PROGRAM PRG_SysPulses
VAR 
// 50% Duty Cycle
	fbXO_250Hz    		:FB_Pulse;	//Correct at 2ms tick
	fbXO_50Hz     		:FB_Pulse;	//Correct at 2ms tick
	fbXO_10Hz			:FB_Pulse;	//Correct at 2ms tick
	fbXO_5Hz			:FB_Pulse;	//Correct at 2ms tick
	fbXO_2Hz			:FB_Pulse;	//Correct at 2ms tick	
	fbXO_1Hz			:FB_Pulse;	//Correct at 2ms tick
	fbXO_05Hz			:FB_Pulse;	//Correct at 2ms tick
	// Frictions
	fbXO_1p85Hz			:FB_Pulse;	//Correct at 2ms tick
	fbXO_1p52Hz			:FB_Pulse;	//Correct at 2ms tick
	fbXO_1p33Hz			:FB_Pulse;	//Correct at 2ms tick
	fbXO_1p19Hz			:FB_Pulse;	//Correct at 2ms tick	
	
// 70/30 Duty Cycle
	fbXO_1Hz_7030		:FB_Pulse;	//Correct at 2ms tick
	
// 80/20 Duty Cycle
	fbXO_1Hz_8020		:FB_Pulse;	//Correct at 2ms tick
//-----------------------------------------------oldschoo1		
END_VAR

(*** Oscilator Pulse Generators at 2ms tick ***)

// 50% Duty Cycle
	fbXO_250Hz(
		bEnable				:=	TRUE,
		tPulseOn			:=	T#2MS,
		tPulseOff			:=	T#2MS,
		bFlash				=>	bFlash250Hz);
	fbXO_50Hz( 
		bEnable	    		:=	TRUE,
		tPulseOn			:=	T#10MS,
		tPulseOff			:=	T#10MS,
		bFlash				=>	bFlash50Hz);
	fbXO_10Hz(
		bEnable				:=	TRUE,
		tPulseOn			:=	T#50MS,
		tPulseOff			:=	T#50MS,
		bFlash				=>	bFlash10Hz);
	fbXO_5Hz(
		bEnable				:=	TRUE,
		tPulseOn			:=	T#100MS,
		tPulseOff			:=	T#100MS,
		bFlash				=>	bFlash5Hz);
	fbXO_2Hz(
		bEnable				:=	TRUE,
		tPulseOn			:=	T#250MS,
		tPulseOff			:=	T#250MS,
		bFlash				=>	bFlash2Hz);
	fbXO_1Hz(
		bEnable				:=	TRUE,
		tPulseOn			:=	T#500MS,
		tPulseOff			:=	T#500MS,
		bFlash				=>	bFlash1Hz);	
	fbXO_05Hz(
		bEnable				:=	TRUE,
		tPulseOn			:=	T#1000MS,
		tPulseOff			:=	T#1000MS,
		bFlash				=>	bFlash05Hz);
//Frictions
	fbXO_1p85Hz(
		bEnable				:=	TRUE,
		tPulseOn			:=	T#270MS,
		tPulseOff			:=	T#270MS,
		bFlash				=>	bFlash1p85Hz);
	fbXO_1p52Hz(
		bEnable				:=	TRUE,
		tPulseOn			:=	T#330MS,
		tPulseOff			:=	T#330MS,
		bFlash				=>	bFlash1p52Hz);
	fbXO_1p33Hz(
		bEnable				:=	TRUE,
		tPulseOn			:=	T#376MS,
		tPulseOff			:=	T#376MS,
		bFlash				=>	bFlash1p33Hz);
	fbXO_1p19Hz(
		bEnable				:=	TRUE,
		tPulseOn			:=	T#416MS,
		tPulseOff			:=	T#416MS,
		bFlash				=>	bFlash1p2Hz);
		
// 70/30 Duty Cycle
	fbXO_1Hz_7030(
		bEnable				:=	TRUE,
		tPulseOn			:=	T#700MS,
		tPulseOff			:=	T#300MS,
		bFlash				=>	bFlash1Hz_7030);
		
// 80/20 Duty Cycle
	fbXO_1Hz_8020(
		bEnable				:=	TRUE,
		tPulseOn			:=	T#800MS,
		tPulseOff			:=	T#200MS,
		bFlash				=>	bFlash1Hz_8020);
//-----------------------------------------------oldschoo1

END_PROGRAM

(* stored: Version 1.1.0.1, ProductVersion 3.1.4024.12
   POU PRG_SysPulses: Id {c28f8fa5-65be-490b-ad96-143277b2a36f}, SpecialFunc None *)
